INTERFACE I_Mode

PROPERTY Mode : E_Mode
GET
END_GET
END_PROPERTY

END_INTERFACE

(* stored: Version 1.1.0.1
   Itf I_Mode: Id {b2658bf8-f506-4366-a44a-b5e7bb4c4ce0}
   Property Mode: Id {77adbbc3-73f0-48e2-9c18-4e644011df58}
   Get Get: Id {c145dfd3-f062-45a3-beef-fb9b527435c9} *)
